(* CoDeSys 2.3.9.48 project: TcpUdp.pro *)
(* Libraries: SysLibSockets.lib*2.6.14 13:06:08, Standard.lib*2.6.14 11:37:46, SYSLIBCALLBACK.LIB*2.6.14 13:06:08 *)

(* Task configuration *)
TASK MainTask (PRIORITY := 10, INTERVAL := T#100ms);
	PLC_PRG();
END_TASK
TASK ServerTask (PRIORITY := 5, INTERVAL := T#10ms);
	TCPServer();
END_TASK
TASK ClientTask (PRIORITY := 3, INTERVAL := T#10ms);
	TCPClient();
END_TASK
TASK ConsumerTask (PRIORITY := 12, INTERVAL := T#10ms);
	UDPConsumer();
END_TASK
TASK ProducerTask (PRIORITY := 8, INTERVAL := T#10ms);
	UDPProducer();
END_TASK

(* Data type *)
TYPE CLIENT_ACCEPT :
STRUCT
	diSocket:DINT;
	stIPAddress:STRING(20);
END_STRUCT
END_TYPE

(* Data type *)
TYPE CLIENT_REPLY :
STRUCT
	diBytesReceived:DINT;
	stIPAddressTransmitter:STRING(20);
END_STRUCT
END_TYPE

(* POU PLC_PRG, ST *)
PROGRAM PLC_PRG
VAR
	bInit:BOOL;
END_VAR
IF NOT bInit THEN
	SysCallbackRegister(INDEXOF(ResetCallback), EVENT_BEFORE_RESET);
	bInit := TRUE;
END_IF
END_PROGRAM

(* POU ResetCallback, ST *)
FUNCTION ResetCallback : DWORD
VAR_INPUT
	dwEvent:DWORD;
	dwFilter:DWORD;
	dwOwner:DWORD;
END_VAR
VAR
END_VAR
IF dwEvent = EVENT_BEFORE_RESET THEN
	IF TCPServer.diSocket <> -1 THEN
		SysSockClose(TCPServer.diSocket);
	END_IF
	IF (TCPServer.Client.diSocket <> -1) THEN
		SysSockClose(TCPServer.Client.diSocket);
	END_IF
	IF TCPClient.diSocket <> -1 THEN
		SysSockClose(TCPClient.diSocket);
	END_IF
	IF UDPProducer.diSendSocket <> -1 THEN
		SysSockClose(UDPProducer.diSendSocket);
	END_IF
	IF UDPConsumer.diRecvSocket <> -1 THEN
		SysSockClose(UDPConsumer.diRecvSocket);
	END_IF
END_IF
END_FUNCTION

(* POU TCPServer, ST *)
PROGRAM TCPServer
VAR
	diSocket : DINT := -1;
	iPort : INT:=4444;
	Client : CLIENT_ACCEPT := (diSocket := -1);
	bySend : ARRAY[0..10] OF BYTE := 0,1,2,3,4,5,6,7,8,9,10;
	byRecv : ARRAY[0..10] OF BYTE;
	Reply : CLIENT_REPLY;
	bCloseClient: BOOL;
	bActive: BOOL;
END_VAR
IF bActive THEN
	IF diSocket = -1 THEN
		diSocket := TcpServerOpenSocket(iPort, 10, 1000);
	END_IF

	IF  Client.diSocket = -1 THEN
		Client := TcpServerWaitForConnect(diSocket, 4);
	END_IF

	IF  Client.diSocket <> -1 THEN
		TcpSendData(Client.diSocket, ADR(bySend), SIZEOF(bySend), 1);
		(*TcpReceiveData(Client.diSocket, ADR(byRecv), SIZEOF(byRecv), 5);*)
	END_IF

	IF bCloseClient THEN
		bCloseClient := FALSE;
		SysSockClose(diSocket:=Client.diSocket);
		Client.diSocket := -1;
	END_IF
END_IF
END_PROGRAM

(* POU Tcp specific/TcpServerOpenSocket, ST *)
FUNCTION TcpServerOpenSocket : DINT
(*	Open a TCP server socket.
	Return:	Main Socket Id
*)
VAR_INPUT
	iPort:INT;						(* Port number *)
	diMaxConnections:DINT;		(* Max possible client connections of the server *)
	diMaxDataSize:DINT;			(* Max size of data to transmitt; if size = 0 default values are used *)
END_VAR
VAR
	diSocket:DINT;
	bResult:BOOL;
	sa:SOCKADDRESS;
	bOptNoDelay:BOOL;
	lOptLinger:SOCKET_LINGER;
END_VAR
diSocket:=SysSockCreate(SOCKET_AF_INET, SOCKET_STREAM, 0);
IF diSocket <> SOCKET_INVALID THEN
(*
	IF diMaxDataSize <> 0 THEN
		SysSockSetOption(diSocket, SOCKET_SOL, SOCKET_SO_SNDBUF, ADR(diMaxDataSize), SIZEOF(diMaxDataSize));
		SysSockSetOption(diSocket, SOCKET_SOL, SOCKET_SO_RCVBUF, ADR(diMaxDataSize), SIZEOF(diMaxDataSize));
	END_IF
	lOptLinger.l_onoff:=0;
	lOptLinger.l_linger:=0;
	SysSockSetOption(diSocket,	SOCKET_SOL, SOCKET_SO_LINGER, ADR(lOptLinger), SIZEOF(lOptLinger));
	bOptNoDelay:=TRUE;
	SysSockSetOption(diSocket,	SOCKET_IPPROTO_TCP, SOCKET_TCP_NODELAY, ADR(bOptNoDelay), SIZEOF(bOptNoDelay));
*)

	sa.sin_family:=SOCKET_AF_INET;
	sa.sin_addr:=SOCKET_INADDR_ANY;
	sa.sin_port:=SysSockHtons(iPort);
	bResult:=SysSockBind(diSocket, ADR(sa), SIZEOF(sa));
	IF bResult = FALSE THEN
		diSocket:=SOCKET_INVALID;
	ELSE
		bResult:=SysSockListen(diSocket, diMaxConnections);
		IF bResult = FALSE THEN
			diSocket:=SOCKET_INVALID;
		END_IF
	END_IF
END_IF
TcpServerOpenSocket:=diSocket;
END_FUNCTION

(* POU Tcp specific/TcpServerWaitForConnect, ST *)
FUNCTION TcpServerWaitForConnect : CLIENT_ACCEPT
(*	Wait for a TCP client to connect.
	ATTENTION:  Function is blocking, until a client tries to connect!
	Return:	diSocket : Socket Id for connection session
				stIPAddress : IP-Address of connected client
*)
VAR_INPUT
	diServerSocket:DINT;
	diTimeout : DINT;	(* Timeout in seconds *)
END_VAR
VAR
	sa:SOCKADDRESS;
	ia:INADDR;
	diSize:DINT;
	fdRead: SOCKET_FD_SET;
	fdWrite:SOCKET_FD_SET;
	fdExcept:SOCKET_FD_SET;
	tvTimeout:SOCKET_TIMEVAL;
END_VAR
tvTimeout.tv_sec := diTimeout ;
tvTimeout.tv_usec := 0;
fdRead.fd_count := 1;
fdRead.fd_array[0] := diServerSocket;
IF (SysSockSelect(SOCKET_FD_SETSIZE, ADR(fdRead), 0, 0, ADR(tvTimeout)) > 0) THEN
	diSize:=SIZEOF(sa);
	TcpServerWaitForConnect.diSocket:=SysSockAccept(diServerSocket, ADR(sa), ADR(diSize));
	ia.S_addr:=DINT_TO_DWORD(sa.sin_addr);
	SysSockInetNtoa(ia, TcpServerWaitForConnect.stIPAddress, SIZEOF(TcpServerWaitForConnect.stIPAddress));
ELSE
	TcpServerWaitForConnect.diSocket := -1;
END_IF
END_FUNCTION

(* POU Tcp specific/TcpSendData, ST *)
FUNCTION TcpSendData : DINT
(*	Send data via TCP socket.
	Return:	Number of bytes sent
*)
VAR_INPUT
	diSocket:DINT;		(* Socket Id *)
	pbyData:DWORD;		(* Address of data buffer *)
	diDataSize:DINT;		(* Size of data to send *)
	diTImeout : DINT;		(* Timeout in seconds *)
END_VAR
VAR
	fdWrite:SOCKET_FD_SET;
	tvTimeout:SOCKET_TIMEVAL;
END_VAR
tvTimeout.tv_sec := diTimeout ;
tvTimeout.tv_usec := 0;
fdWrite.fd_count := 1;
fdWrite.fd_array[0] := diSocket;
IF (SysSockSelect(SOCKET_FD_SETSIZE, 0, ADR(fdWrite), 0, ADR(tvTimeout)) > 0) THEN
	TcpSendData:=SysSockSend(diSocket, pbyData, diDataSize, 0);
END_IF
END_FUNCTION

(* POU TCPClient, ST *)
PROGRAM TCPClient
VAR
	diSocket : DINT := -1;
	iPort : INT:=4444;
	stDestIPAddress : STRING := '127.0.0.1';
	bySend : ARRAY[0..10] OF BYTE := 0,1,2,3,4,5,6,7,8,9,10;
	byRecv : ARRAY[0..10] OF BYTE;
	bCloseClient: BOOL;
	bActive: BOOL;
END_VAR
IF bActive THEN
	IF diSocket = -1 THEN
		diSocket := TcpClientOpenSocket(iPort, stDestIPAddress, 1000);
	END_IF

	IF  diSocket <> -1 THEN
		TcpReceiveData(diSocket, ADR(byRecv), SIZEOF(byRecv), 5);
		TcpSendData(diSocket, ADR(bySend), SIZEOF(bySend), 1);
	END_IF

	IF bCloseClient THEN
		bCloseClient := FALSE;
		SysSockClose(diSocket:=diSocket);
		diSocket := -1;
	END_IF
END_IF
END_PROGRAM

(* POU Tcp specific/TcpClientOpenSocket, ST *)
FUNCTION TcpClientOpenSocket : DINT
(*	Open TCP client socket to connect to server.
	Return:	Socket-Id for connection session
*)
VAR_INPUT
	iPort:INT;					(* Port number of TCP socket to open *)
	stIPAddress:STRING;		(* IP-Address of server to connect to *)
	diMaxDataSize:DINT;		(* Max size of data to transmitt; if size = 0 default values are used *)
END_VAR
VAR
	diSocket:DINT;
	bOptNoDelay:BOOL;
	lOptLinger:SOCKET_LINGER;
	bResult:BOOL;
	sa:SOCKADDRESS;
END_VAR
diSocket:=SysSockCreate(SOCKET_AF_INET, SOCKET_STREAM, 0);
IF diSocket <> SOCKET_INVALID THEN
	SysSockSetOption(diSocket, SOCKET_SOL, SOCKET_SO_SNDBUF, ADR(diMaxDataSize), SIZEOF(diMaxDataSize));
	SysSockSetOption(diSocket, SOCKET_SOL, SOCKET_SO_RCVBUF, ADR(diMaxDataSize), SIZEOF(diMaxDataSize));
	lOptLinger.l_onoff:=0;
	lOptLinger.l_linger:=0;
	SysSockSetOption(diSocket,	SOCKET_SOL, SOCKET_SO_LINGER, ADR(lOptLinger), SIZEOF(lOptLinger));
	bOptNoDelay:=TRUE;
	SysSockSetOption(diSocket,	SOCKET_IPPROTO_TCP, SOCKET_TCP_NODELAY, ADR(bOptNoDelay), SIZEOF(bOptNoDelay));

	sa.sin_family:=SOCKET_AF_INET;
	sa.sin_addr:=GetIPAddress(stIPAddress);
	IF sa.sin_addr <> SOCKET_INADDR_NONE THEN
		sa.sin_port:=SysSockHtons(iPort);
		IF SysSockConnect(diSocket, ADR(sa), SIZEOF(sa)) = FALSE THEN
			SysSockClose(diSocket);
			diSocket:=SOCKET_INVALID;
		END_IF
	ELSE
		SysSockClose(diSocket);
		diSocket:=SOCKET_INVALID;
	END_IF
END_IF
TcpClientOpenSocket:=diSocket;
END_FUNCTION

(* POU GetIPAddress, ST *)
FUNCTION GetIPAddress : DINT
(*	Convert IP-Address from string to address.
	Return:	IP-address
 *)
VAR_INPUT
	stIPAddress:STRING;		(* IP-address or computer name *)
END_VAR
VAR
	diIPAddress:DINT;
END_VAR
diIPAddress := SysSockInetAddr(stIPAddress);
IF diIPAddress = SOCKET_INADDR_NONE THEN
	diIPAddress := SysSockGetHostByName(ADR(stIPAddress));
END_IF
GetIPAddress:=diIPAddress;
END_FUNCTION

(* POU Tcp specific/TcpReceiveData, ST *)
FUNCTION TcpReceiveData : DINT
(*	Receive data from a tcp socket.
	Return:	Number of bytes received
*)
VAR_INPUT
	diSocket:DINT;		(* Socket Id *)
	pbyData:DWORD;		(* Address of data buffer *)
	diDataSize:DINT;		(* Size of data to send *)
	diTImeout : DINT;		(* Timeout in seconds *)
END_VAR
VAR
	fdRead:SOCKET_FD_SET;
	tvTimeout:SOCKET_TIMEVAL;
END_VAR
tvTimeout.tv_sec := diTimeout ;
tvTimeout.tv_usec := 0;
fdRead.fd_count := 1;
fdRead.fd_array[0] := diSocket;
IF (SysSockSelect(SOCKET_FD_SETSIZE, ADR(fdRead), 0, 0, ADR(tvTimeout)) > 0) THEN
	TcpReceiveData:=SysSockRecv(diSocket, pbyData, diDataSize, 0);
END_IF
END_FUNCTION

(* POU UDPProducer, ST *)
PROGRAM UDPProducer
VAR
	diSendSocket : DINT;
	iPort : INT:=4444;
	stDestIPAddress : STRING := '127.0.0.1';
	diRecvSocket: DINT;
	bySend : ARRAY[0..10] OF BYTE := 0,1,2,3,4,5,6,7,8,9,10;
	bSent: BOOL;
	bActive: BOOL;
END_VAR
IF bActive THEN
	IF diSendSocket = 0 THEN
		diSendSocket := UdpOpenSendSocket(iPort);
	END_IF
	
	IF diSendSocket > 0 AND bSent THEN
		bSent := FALSE;
		UdpSendData(diSendSocket, iPort, stDestIPAddress, ADR(bySend), SIZEOF(bySend));
	END_IF
END_IF
END_PROGRAM

(* POU Udp specific/UdpOpenSendSocket, ST *)
FUNCTION UdpOpenSendSocket : DINT
(*	Open socket to send data via UDP.
	Return:	Socket Id
*)
VAR_INPUT
	iPort:INT;		(* Port number *)
END_VAR
VAR
	diSocket:DINT;
	diOption:DINT;
END_VAR
diSocket:=SysSockCreate(SOCKET_AF_INET, SOCKET_DGRAM, 0);
IF diSocket = SOCKET_INVALID THEN
	UdpOpenSendSocket:=SOCKET_INVALID;
ELSE
(*
	diOption:=1;
	IF SysSockSetOption(diSocket, SOCKET_SOL, SOCKET_SO_BROADCAST, ADR(diOption), SIZEOF(diOption)) = FALSE THEN
		UdpOpenSendSocket:=SOCKET_INVALID;
	ELSE
*)
		UdpOpenSendSocket:=diSocket;
(*
	END_IF
*)
END_IF
END_FUNCTION

(* POU Udp specific/UdpSendData, ST *)
FUNCTION UdpSendData : DINT
(* Function to send data via UDP protocol.
	Return:	Number of bytes realy sent
*)	
VAR_INPUT
	diSocket:DINT;		(* Socket Id *)
	iPort:INT;				(* Port number, to send data *)
	stIPAddress:STRING;		(* IP-address or name *)
	pbyData:DWORD;		(* Address of data buffer *)
	diDataSize:DINT;		(* Size of data to send *)
END_VAR
VAR
	sa:SOCKADDRESS;
END_VAR
sa.sin_family:=SOCKET_AF_INET;
IF stIPAddress <> '' THEN
	sa.sin_addr:=GetIPAddress(stIPAddress);
ELSE
	sa.sin_addr:=SOCKET_INADDR_BROADCAST;
END_IF
sa.sin_port:=SysSockHtons(iPort);
UdpSendData:=SysSockSendTo(diSocket, pbyData, diDataSize, 0, ADR(sa), SIZEOF(sa));
END_FUNCTION

(* POU UDPConsumer, ST *)
PROGRAM UDPConsumer
VAR
	iPort : INT:=4444;
	stDestIPAddress : STRING := '127.0.0.1';
	diRecvSocket: DINT;
	byRecv : ARRAY[0..10] OF BYTE;
	Reply : CLIENT_REPLY;
	bActive: BOOL;
END_VAR
IF bActive THEN
	IF diRecvSocket = 0 THEN
		diRecvSocket := UdpOpenReceiveSocket(iPort);
	END_IF
	
	IF diRecvSocket > 0 THEN
		Reply := UdpReceiveData(diRecvSocket, iPort, ADR(byRecv), SIZEOF(byRecv));
	END_IF
END_IF
END_PROGRAM

(* POU Udp specific/UdpOpenReceiveSocket, ST *)
FUNCTION UdpOpenReceiveSocket : DINT
(*	Open socket to receive data via UDP.
	Return:	Socket Id
*)
VAR_INPUT
	iPort:INT;		(* Port number *)
END_VAR
VAR
	diSocket:DINT;
	bResult:BOOL;
	sa:SOCKADDRESS;
END_VAR
diSocket:=SysSockCreate(SOCKET_AF_INET, SOCKET_DGRAM, 0);
sa.sin_family:=SOCKET_AF_INET;
sa.sin_addr:=SOCKET_INADDR_ANY;
sa.sin_port:=SysSockHtons(iPort);
bResult:=SysSockBind(diSocket, ADR(sa), SIZEOF(sa));
IF bResult = FALSE THEN
	diSocket:=SOCKET_INVALID;
END_IF
UdpOpenReceiveSocket:=diSocket;
END_FUNCTION

(* POU Udp specific/UdpReceiveData, ST *)
FUNCTION UdpReceiveData : CLIENT_REPLY
(* Function to receive data via UDP protocol.
	Return:	diBytesReceived:Number of bytes received
				stIPAddressTransmitter: IP-address of client, that sent the data
 *)	
VAR_INPUT
	diSocket:DINT;		(* Socket Id *)
	iPort:INT;				(* Port number, to send data *)
	pbyData:DWORD;		(* Address of data buffer *)
	diDataSize:DINT;		(* Size of data to send *)
END_VAR
VAR
	sa:SOCKADDRESS;
	ia:INADDR;
	saSize:DINT;
END_VAR
UdpReceiveData.diBytesReceived:=SysSockRecvFrom(diSocket, pbyData, diDataSize, 0, ADR(sa), SIZEOF(sa));
ia.S_addr:=DINT_TO_DWORD(sa.sin_addr);
SysSockInetNtoa(ia, UdpReceiveData.stIPAddressTransmitter, SIZEOF(UdpReceiveData.stIPAddressTransmitter));
END_FUNCTION

(* POU ConvertPAddressToString, ST *)
FUNCTION ConvertPAddressToString : STRING
(*	Convert the IP-Address to a string in dot-notation, e.g. '192.168.100.2' .
	Return:	IP-address
 *)
VAR_INPUT
	diIPAddress:DINT;
END_VAR
VAR
	iadr:INADDR;
	stIP:STRING;
END_VAR
iadr.S_addr := diIPAddress;
SysSockInetNtoa(iadr, stIP, SIZEOF(stIP));
ConvertPAddressToString:=stIP;
END_FUNCTION

(* POU GetReceiveDataSize, ST *)
FUNCTION GetReceiveDataSize : DINT
(* Function to get received number of bytes in socket, without removing it from the socket.
	Return:	Number of bytes received
 *)	
VAR_INPUT
	diSocket	: DINT;		(* Socket Id *)
END_VAR
VAR
	diParameter:DINT;
END_VAR
diParameter:=0;
IF SysSockIoctl(diSocket, SOCKET_FIONREAD, ADR(diParameter)) = 1 THEN
	GetReceiveDataSize := diParameter;
ELSE
	GetReceiveDataSize := 0;
END_IF
END_FUNCTION
